{attribute addProperty BoxType "EL5122-0000-0016"}
{attribute addProperty Id "Latch_extern_validBIT10.1252Set_counter_doneBIT10.1253Counter_underflowBIT10.1254Counter_overflowBIT10.1255Status_of_input_ABIT10.1259Status_of_input_BBIT10.12510Status_of_input_gateBIT10.12512DiagBIT10.12513TxPDO_StateBIT10.12514Input_cycle_counter_BIT_0BIT10.12515Input_cycle_counter_BIT_1BIT10.12515Software_gate_validBIT10.12517Counter_value_out_of_rangeBIT10.12521"}
{attribute addProperty CRC "938646721"}
{attribute addProperty SizeInBites "32"}
{attribute addProperty SizeInBytes "4"}
TYPE Status_37F29CC1 :
STRUCT
	{attribute 'hide'}
	reserve_1 : BIT;
	{attribute addProperty Name "Latch_extern_valid"}
	Latch_extern_valid : BIT;
	{attribute addProperty Name "Set_counter_done"}
	Set_counter_done : BIT;
	{attribute addProperty Name "Counter_underflow"}
	Counter_underflow : BIT;
	{attribute addProperty Name "Counter_overflow"}
	Counter_overflow : BIT;
	{attribute 'hide'}
	reserve_2 : BIT;
	{attribute 'hide'}
	reserve_3 : BIT;
	{attribute 'hide'}
	reserve_4 : BIT;
	{attribute addProperty Name "Status_of_input_A"}
	Status_of_input_A : BIT;
	{attribute addProperty Name "Status_of_input_B"}
	Status_of_input_B : BIT;
	{attribute 'hide'}
	reserve_5 : BIT;
	{attribute addProperty Name "Status_of_input_gate"}
	Status_of_input_gate : BIT;
	{attribute addProperty Name "Diag"}
	Diag : BIT;
	{attribute addProperty Name "TxPDO_State"}
	TxPDO_State : BIT;
	{attribute addProperty Name "Input_cycle_counter"}
	Input_cycle_counter_BIT_0 : BIT;
	{attribute addProperty Name "Input_cycle_counter"}
	Input_cycle_counter_BIT_1 : BIT;
	{attribute addProperty Name "Software_gate_valid"}
	Software_gate_valid : BIT;
	{attribute 'hide'}
	reserve_6 : BIT;
	{attribute 'hide'}
	reserve_7 : BIT;
	{attribute 'hide'}
	reserve_8 : BIT;
	{attribute addProperty Name "Counter_value_out_of_range"}
	Counter_value_out_of_range : BIT;
	{attribute 'hide'}
	reserve_9_BIT_0 : BIT;
	{attribute 'hide'}
	reserve_9_BIT_1 : BIT;
	{attribute 'hide'}
	reserve_9_BIT_2 : BIT;
	{attribute 'hide'}
	reserve_10 : BYTE;
END_STRUCT
END_TYPE

(* stored: Version 1.2.0.0, ProductVersion 3.1.4024.9
   DUT Status_37F29CC1: Id {16838876-1f2c-4bbe-9bc9-9379ace367bb} *)
